FUNCTION_BLOCK TcoComponentTestContext EXTENDS TcoCore._internals_TcoContext
VAR
    _sut : TestComponent(THIS^);
    {attribute addProperty Name "--Some IO signal"}
    _signal : BOOL;
END_VAR

METHOD PROTECTED Main
CASE _testId OF
    eTcoComponentTests.GetSignalInfo:
        _sut(_signal := _signal);
END_CASE
END_METHOD

END_FUNCTION_BLOCK

(* stored: Version 1.1.0.1
   POU TcoComponentTestContext: Id {d9b91383-f3ba-02bf-3371-fb3da801fc57}, SpecialFunc None
   Method Main: Id {d6ce3f3d-729e-0c45-285b-5f1b5d239c1e} *)
